// SIMATIC S7-200 SMART project (STEP 7-Micro/WIN SMART), CPU SR20

SYMBOL_TABLE Table 1
                 VW1      // LineSetTimeHMI
                 M13.0    // Line1repeat1
                 M9.0     // Line1OneLap
                 VW80     // Line2SetTimeHMI
END_SYMBOL_TABLE

SYMBOL_TABLE System Symbols
Clock_1s         SM0.5    // Clock pulse that is ON for 0.5 s, OFF for 0.5 s, for a duty cycle time of 1 s.
END_SYMBOL_TABLE

ORGANIZATION_BLOCK MAIN:OB1
TITLE=Program Comments
BEGIN
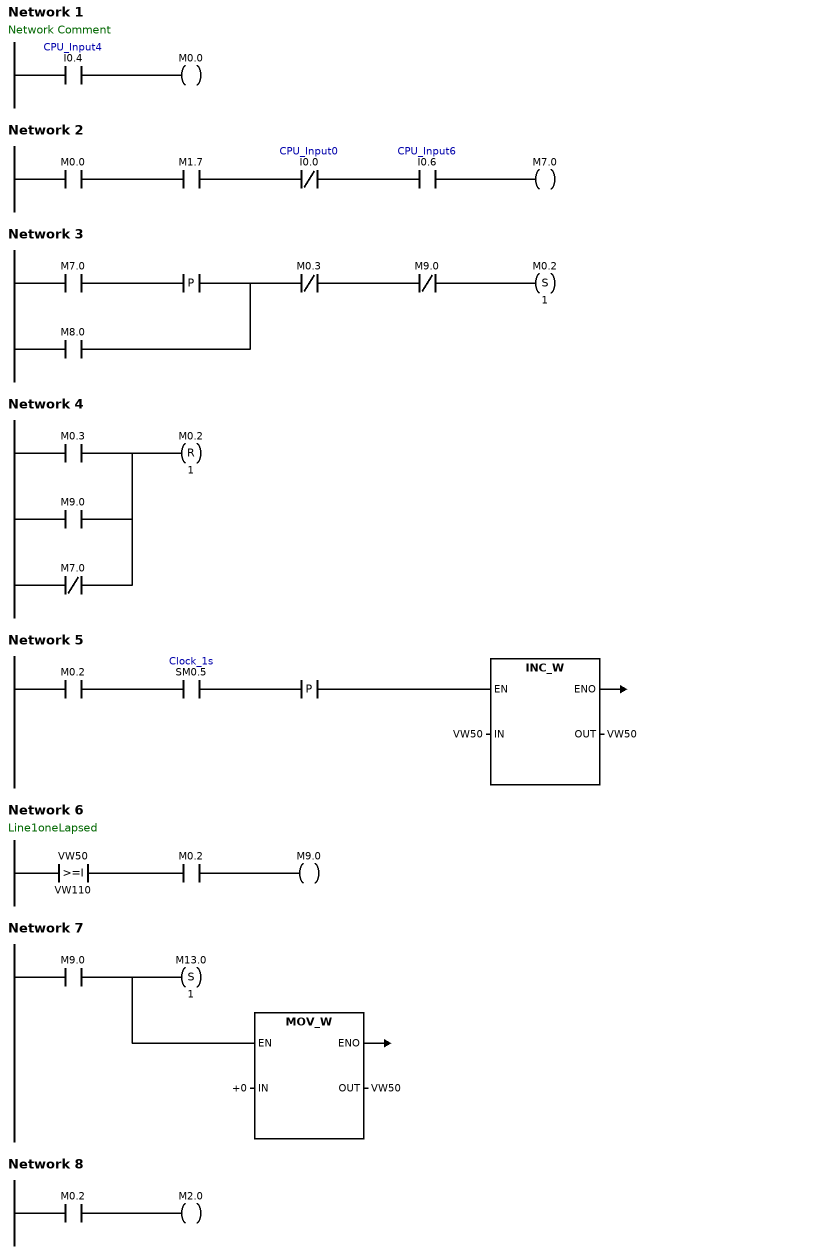
Network 1
// Network Comment
LD     CPU_Input4:I0.4
=      M0.0
Network 2
LD     M0.0
A      M1.7
AN     CPU_Input0:I0.0
A      CPU_Input6:I0.6
=      M7.0
Network 3
LD     M7.0
EU
O      M8.0
AN     M0.3
AN     M9.0
S      M0.2, 1
Network 4
LD     M0.3
O      M9.0
ON     M7.0
R      M0.2, 1
Network 5
//  
LD     M0.2
A      Clock_1s:SM0.5
EU
INCW   VW50
Network 6
// Line1oneLapsed
LDW>=  VW50, VW110
A      M0.2
=      M9.0
Network 7
LD     M9.0
S      M13.0, 1
MOVW   +0, VW50
Network 8
LD     M0.2
=      M2.0
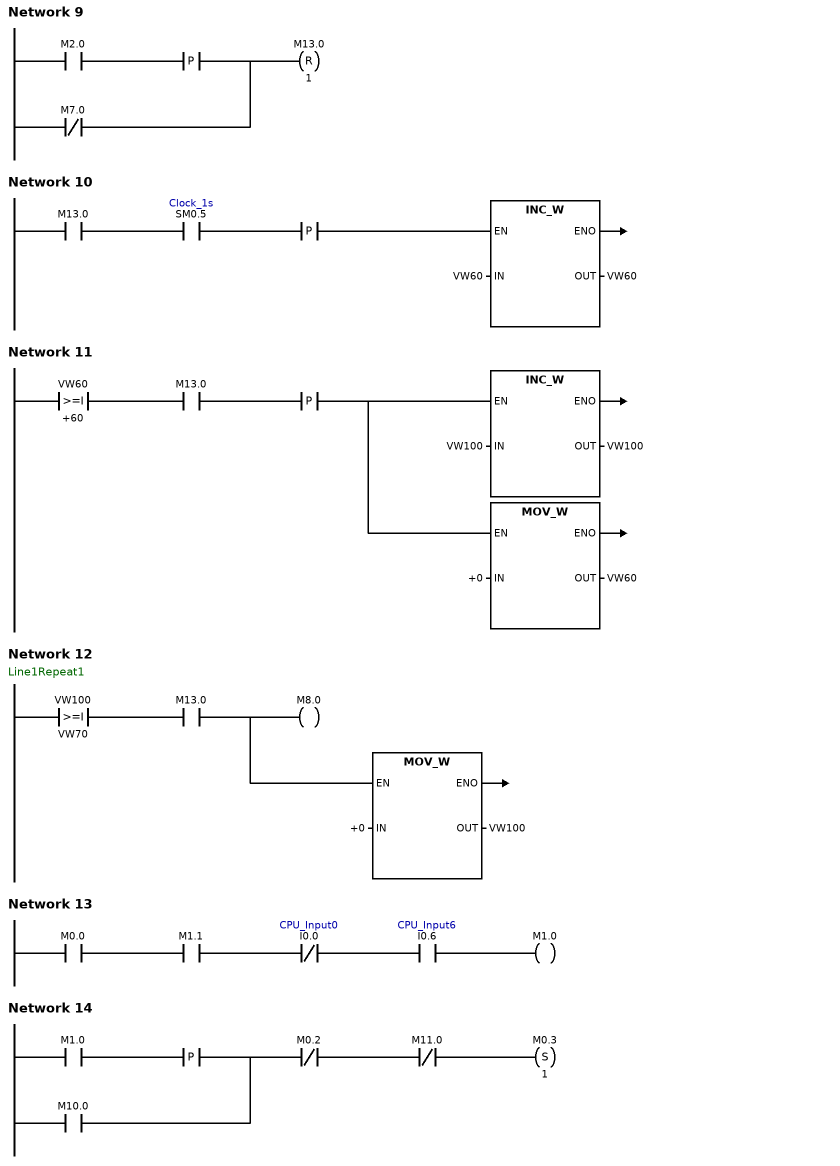
Network 9
LD     M2.0
EU
ON     M7.0
R      M13.0, 1
Network 10
LD     M13.0
A      Clock_1s:SM0.5
EU
INCW   VW60
Network 11
LDW>=  VW60, +60
A      M13.0
EU
INCW   VW100
MOVW   +0, VW60
Network 12
// Line1Repeat1
LDW>=  VW100, VW70
A      M13.0
=      M8.0
MOVW   +0, VW100
Network 13
LD     M0.0
A      M1.1
AN     CPU_Input0:I0.0
A      CPU_Input6:I0.6
=      M1.0
Network 14
LD     M1.0
EU
O      M10.0
AN     M0.2
AN     M11.0
S      M0.3, 1
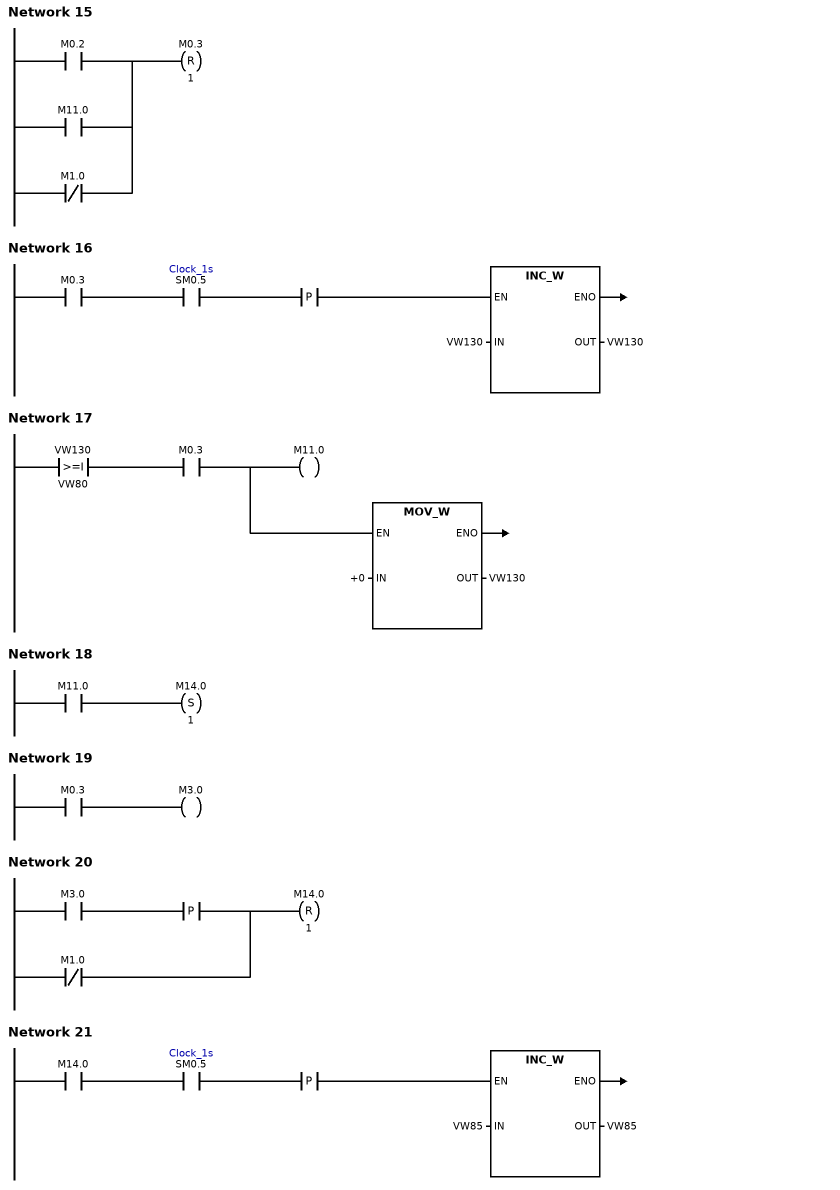
Network 15
LD     M0.2
O      M11.0
ON     M1.0
R      M0.3, 1
Network 16
LD     M0.3
A      Clock_1s:SM0.5
EU
INCW   VW130
Network 17
LDW>=  VW130, VW80
A      M0.3
=      M11.0
MOVW   +0, VW130
Network 18
LD     M11.0
S      M14.0, 1
Network 19
LD     M0.3
=      M3.0
Network 20
LD     M3.0
EU
ON     M1.0
R      M14.0, 1
Network 21
LD     M14.0
A      Clock_1s:SM0.5
EU
INCW   VW85
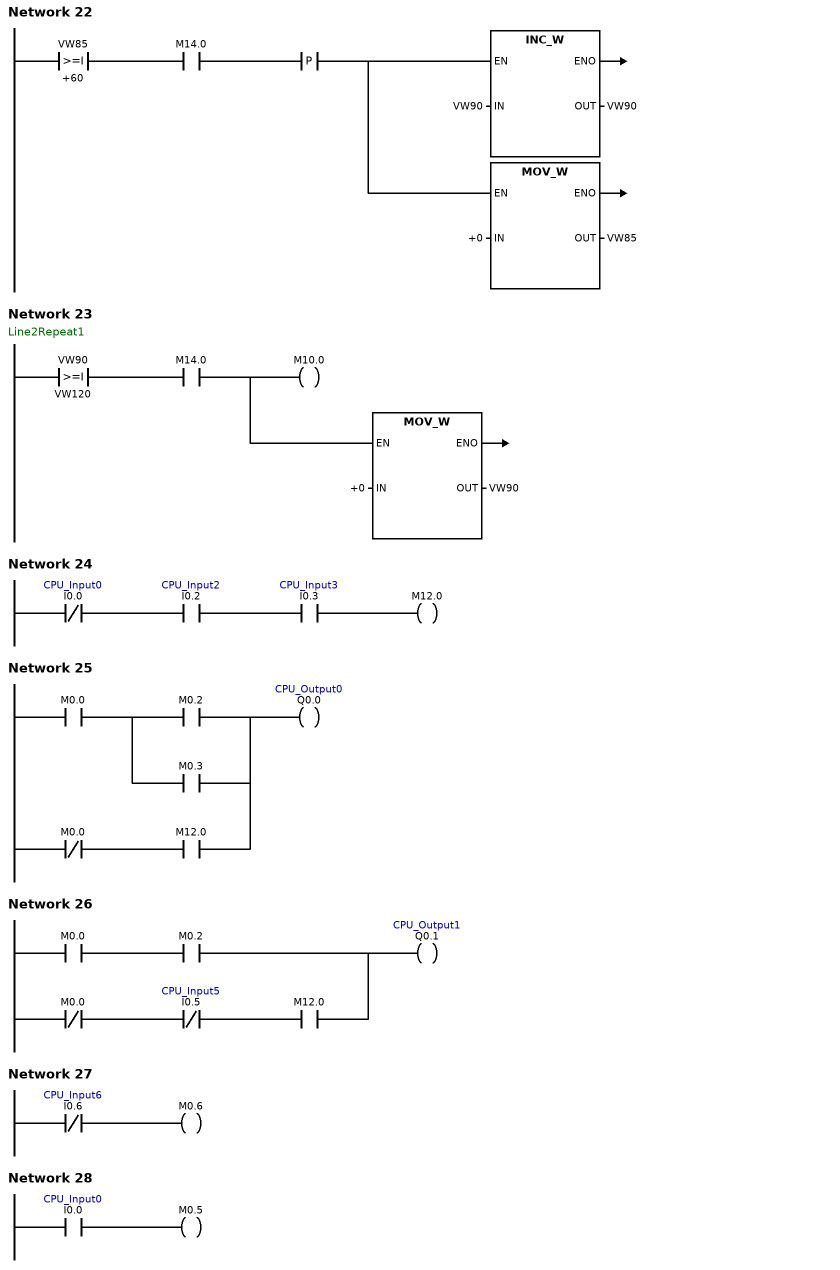
Network 22
LDW>=  VW85, +60
A      M14.0
EU
INCW   VW90
MOVW   +0, VW85
Network 23
// Line2Repeat1
LDW>=  VW90, VW120
A      M14.0
=      M10.0
MOVW   +0, VW90
Network 24
LDN    CPU_Input0:I0.0
A      CPU_Input2:I0.2
A      CPU_Input3:I0.3
=      M12.0
Network 25
LD     M0.0
LD     M0.2
O      M0.3
ALD
LDN    M0.0
A      M12.0
OLD
=      CPU_Output0:Q0.0
Network 26
LD     M0.0
A      M0.2
LDN    M0.0
AN     CPU_Input5:I0.5
A      M12.0
OLD
=      CPU_Output1:Q0.1
Network 27
LDN    CPU_Input6:I0.6
=      M0.6
Network 28
LD     CPU_Input0:I0.0
=      M0.5
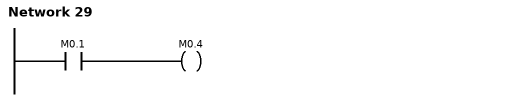
Network 29
LD     M0.1
=      M0.4
END_ORGANIZATION_BLOCK
